(* IEC 61131-3 sources: canworks/test/cia402, 6 files *)

(* ---- drive_model.st ---- *)
(*
 * A CiA 402 drive for the ST tests (test/cia402/run.sh): the power state
 * machine (CiA 402 figure "state machine"), profile position (mode 1),
 * profile velocity (mode 3), homing (mode 6, method 35: the current
 * position is home) and the cyclic synchronous modes (8 position, 9
 * velocity, 10 torque: the set-point of each call is applied, as on one
 * SYNC), with halt (controlword bit 8) and a fault input. A mode that
 * ModesSupported (0x6502 bits) does not list is not taken: 0x6061 keeps the
 * old mode. One call is one cycle of Dt. test/drive/cia402_slave.hpp plays
 * the profile modes on a CAN bus.
 *
 * Statusword bits: 0 ready to switch on, 1 switched on, 2 operation enabled,
 * 3 fault, 4 voltage enabled, 5 quick stop (1 = not active), 6 switch on
 * disabled, 9 remote, 10 target reached, 12 set-point acknowledge / speed
 * zero / homing attained (by mode), 14 standstill (the bit the editor's
 * motion library reads as standstill).
 *)
FUNCTION_BLOCK CiA402_Drive
VAR_INPUT
	ControlWord : UINT;
	Modes : SINT;
	TargetPosition : DINT;
	ProfileVelocity : UDINT;
	TargetVelocity : DINT;
	TargetTorque : INT;
	Fault : BOOL;                (* raise a drive fault *)
	Dt : LREAL := 0.01;          (* cycle [s] *)
	ModesSupported : DWORD := DWORD#16#000003A5;  (* 0x6502: modes 1, 3, 6, 8, 9, 10 *)
	TorqueGain : LREAL := 10.0;  (* mode 10: acceleration [counts/s2] per mille of torque *)
END_VAR
VAR_OUTPUT
	StatusWord : UINT;
	ModesDisplay : SINT;
	Position : DINT;
	Velocity : DINT;
	Torque : INT;
	State : INT;                 (* 1 switch on disabled, 2 ready, 3 switched on, 4 enabled, 5 quick stop, 6 fault *)
END_VAR
VAR
	pos : LREAL;
	vel : LREAL;
	target : LREAL;
	cw : WORD;
	lastCw : WORD;
	ack : BOOL;
	homed : BOOL;
	step : LREAL;
END_VAR
	cw := UINT_TO_WORD(ControlWord);
	IF State = 0 THEN
		State := 1;
	END_IF

	(* Power state machine *)
	IF Fault AND State <> 6 THEN
		State := 6;
	ELSIF State = 6 THEN
		IF cw.7 AND NOT lastCw.7 AND NOT Fault THEN
			State := 1;
		END_IF
	ELSIF (cw AND WORD#16#0082) = WORD#16#0000 THEN
		State := 1;                                        (* disable voltage *)
	ELSIF (cw AND WORD#16#0086) = WORD#16#0002 THEN
		IF State = 4 THEN State := 5; ELSE State := 1; END_IF  (* quick stop *)
	ELSIF (cw AND WORD#16#0087) = WORD#16#0006 THEN
		State := 2;                                        (* shutdown *)
	ELSIF (cw AND WORD#16#008F) = WORD#16#0007 THEN
		IF State = 2 OR State = 4 THEN State := 3; END_IF  (* switch on / disable operation *)
	ELSIF (cw AND WORD#16#008F) = WORD#16#000F THEN
		IF State = 3 OR State = 5 THEN State := 4; END_IF  (* enable operation *)
	END_IF

	IF Modes >= SINT#1 AND Modes <= SINT#32 THEN
		IF (SHR(ModesSupported, SINT_TO_INT(Modes) - 1) AND DWORD#1) = DWORD#1 THEN
			ModesDisplay := Modes;
		END_IF
	END_IF
	Torque := 0;
	IF State <> 4 THEN
		vel := 0.0;
		ack := FALSE;
		target := pos;
	ELSIF cw.8 THEN
		vel := 0.0;                                        (* halt *)
	ELSIF ModesDisplay = 1 THEN
		IF cw.4 AND NOT lastCw.4 THEN
			IF cw.6 THEN target := target + DINT_TO_LREAL(TargetPosition);
			ELSE target := DINT_TO_LREAL(TargetPosition); END_IF
			ack := TRUE;
		ELSIF NOT cw.4 THEN
			ack := FALSE;
		END_IF
		step := UDINT_TO_LREAL(ProfileVelocity) * Dt;
		IF ABS(target - pos) <= step THEN
			vel := (target - pos) / Dt;
		ELSIF target > pos THEN
			vel := UDINT_TO_LREAL(ProfileVelocity);
		ELSE
			vel := -UDINT_TO_LREAL(ProfileVelocity);
		END_IF
	ELSIF ModesDisplay = 3 THEN
		vel := DINT_TO_LREAL(TargetVelocity);
	ELSIF ModesDisplay = 8 THEN
		vel := (DINT_TO_LREAL(TargetPosition) - pos) / Dt;   (* CSP: at the set-point after one cycle *)
		target := DINT_TO_LREAL(TargetPosition);
	ELSIF ModesDisplay = 9 THEN
		vel := DINT_TO_LREAL(TargetVelocity);
	ELSIF ModesDisplay = 10 THEN
		vel := vel + INT_TO_LREAL(TargetTorque) * TorqueGain * Dt;
		Torque := TargetTorque;
	ELSIF ModesDisplay = 6 THEN
		vel := 0.0;
		IF cw.4 AND NOT lastCw.4 THEN
			pos := 0.0;                                    (* method 35: here is home *)
			target := 0.0;
			homed := TRUE;
		ELSIF NOT cw.4 THEN
			homed := FALSE;
		END_IF
	ELSE
		vel := 0.0;
	END_IF
	pos := pos + vel * Dt;
	Position := LREAL_TO_DINT(pos);
	Velocity := LREAL_TO_DINT(vel);

	(* Statusword *)
	CASE State OF
		1: StatusWord := 16#0250;   (* switch on disabled, quick stop off, remote *)
		2: StatusWord := 16#0231;
		3: StatusWord := 16#0233;
		4: StatusWord := 16#0237;
		5: StatusWord := 16#0217;
		6: StatusWord := 16#0218;
	END_CASE
	IF vel = 0.0 THEN
		StatusWord := StatusWord OR 16#4000;                (* standstill *)
	END_IF
	IF State = 4 THEN
		IF ModesDisplay = 1 THEN
			IF ack THEN StatusWord := StatusWord OR 16#1000; END_IF
			IF pos = target THEN StatusWord := StatusWord OR 16#0400; END_IF
		ELSIF ModesDisplay = 3 THEN
			IF vel = 0.0 THEN StatusWord := StatusWord OR 16#1000; END_IF
			IF vel = DINT_TO_LREAL(TargetVelocity) THEN StatusWord := StatusWord OR 16#0400; END_IF
		ELSIF ModesDisplay = 6 THEN
			IF homed THEN StatusWord := StatusWord OR 16#1400; END_IF
		ELSIF ModesDisplay >= 8 AND ModesDisplay <= 10 THEN
			StatusWord := StatusWord OR 16#1000;            (* drive follows the command value *)
		END_IF
	END_IF
	lastCw := cw;
END_FUNCTION_BLOCK

(*
 * One bus cycle between a program and a CiA402_Drive: call it with the
 * outputs the program wrote, then copy its outputs into the program's
 * inputs (the test runner does not write VAR_IN_OUT back into a program's
 * located variables, so the test files copy them).
 *)
FUNCTION_BLOCK DriveLink
VAR_INPUT
	ControlWord : UINT;
	Modes : SINT;
	TargetPosition : DINT;
	ProfileVelocity : UDINT;
	TargetVelocity : DINT;
	TargetTorque : INT;
	Fault : BOOL;
	Lost : BOOL;                 (* the node stops answering: inputs hold, status bit FALSE *)
END_VAR
VAR_OUTPUT
	StatusWord : UINT;
	ModesDisplay : SINT;
	Position : DINT;
	Velocity : DINT;
	Torque : INT;
	Online : BOOL;
END_VAR
VAR
	Drive : CiA402_Drive;
END_VAR
	Online := NOT Lost;
	IF NOT Lost THEN
		Drive(ControlWord := ControlWord, Modes := Modes, TargetPosition := TargetPosition,
		      ProfileVelocity := ProfileVelocity, TargetVelocity := TargetVelocity, TargetTorque := TargetTorque,
		      Fault := Fault);
		StatusWord := Drive.StatusWord;
		ModesDisplay := Drive.ModesDisplay;
		Position := Drive.Position;
		Velocity := Drive.Velocity;
		Torque := Drive.Torque;
	END_IF
END_FUNCTION_BLOCK

(* ---- test_axis.st ---- *)
(*
 * The program the project generator writes for config/cia402-drive (its
 * axis `drive` and the bridge call), with the editor's PLCopen motion blocks
 * called on that axis, against the drive model. Run by test/cia402/run.sh.
 * Each cycle: the program's scan, the test's motion block calls (after the
 * bridge, as in a user program), one bus cycle. Time stands still (the test
 * runner advances it only between test statements, not inside a loop), so
 * the library's timeouts never fire; the drive model moves by its own Dt.
 *)
TEST 'MC_Power enables the drive through the CiA 402 state machine'
	VAR
		m : main;
		bus : DriveLink;
		power : MC_Power;
		status : MC_ReadStatus;
		i : INT;
		seenShutdown, seenSwitchOn : BOOL;
	END_VAR
	FOR i := 1 TO 40 DO
		m();
		power(Axis := m.drive, Enable := TRUE);
		bus(ControlWord := m.drive_Controlword, Modes := m.drive_Modes_of_operation,
		    TargetPosition := m.drive_Target_position, ProfileVelocity := m.drive_Profile_velocity,
		    TargetVelocity := m.drive_Target_velocity);
		m.drive_Statusword := bus.StatusWord;
		m.drive_Modes_of_operation_display := bus.ModesDisplay;
		m.drive_Position_actual_value := bus.Position;
		m.drive_Velocity_actual_value := bus.Velocity;
		m.drive_ok := bus.Online;
		IF (m.drive_Controlword AND 16#8F) = 16#06 THEN seenShutdown := TRUE; END_IF
		IF (m.drive_Controlword AND 16#8F) = 16#07 THEN seenSwitchOn := TRUE; END_IF
	END_FOR
	ASSERT_TRUE(seenShutdown, 'drive got Shutdown');
	ASSERT_TRUE(seenSwitchOn, 'drive got Switch on');
	ASSERT_EQ(m.drive_Controlword AND 16#8F, 16#0F, 'drive got Enable operation');
	ASSERT_EQ(bus.Drive.State, 4);
	ASSERT_TRUE(power.Status);
	ASSERT_TRUE(m.drive.bRegulatorRealState);
	status(Axis := m.drive, Enable := TRUE);
	ASSERT_TRUE(status.StandStill);
END_TEST

TEST 'MC_MoveVelocity sets mode 3 and the target velocity'
	VAR
		m : main;
		bus : DriveLink;
		power : MC_Power;
		status : MC_ReadStatus;
		i : INT;
		move : MC_MoveVelocity;
	END_VAR
	FOR i := 1 TO 80 DO
		m();
		power(Axis := m.drive, Enable := TRUE);
		move(Axis := m.drive, Execute := power.Status, Velocity := 1000.0);
		bus(ControlWord := m.drive_Controlword, Modes := m.drive_Modes_of_operation,
		    TargetPosition := m.drive_Target_position, ProfileVelocity := m.drive_Profile_velocity,
		    TargetVelocity := m.drive_Target_velocity);
		m.drive_Statusword := bus.StatusWord;
		m.drive_Modes_of_operation_display := bus.ModesDisplay;
		m.drive_Position_actual_value := bus.Position;
		m.drive_Velocity_actual_value := bus.Velocity;
		m.drive_ok := bus.Online;
	END_FOR
	ASSERT_EQ(m.drive_Modes_of_operation, 3);
	ASSERT_EQ(m.drive_Target_velocity, 1000);
	ASSERT_EQ(m.drive_Velocity_actual_value, 1000);
	ASSERT_TRUE(move.InVelocity);
	status(Axis := m.drive, Enable := TRUE);
	ASSERT_TRUE(status.ContinuousMotion);
	ASSERT_GT(m.drive.fActPosition, 100.0);
END_TEST

TEST 'MC_MoveAbsolute reaches the target in profile position'
	VAR
		m : main;
		bus : DriveLink;
		power : MC_Power;
		status : MC_ReadStatus;
		i : INT;
		move : MC_MoveAbsolute;
		busy : BOOL;
	END_VAR
	FOR i := 1 TO 200 DO
		m();
		power(Axis := m.drive, Enable := TRUE);
		move(Axis := m.drive, Execute := power.Status, Position := 500.0, Velocity := 2000.0);
		bus(ControlWord := m.drive_Controlword, Modes := m.drive_Modes_of_operation,
		    TargetPosition := m.drive_Target_position, ProfileVelocity := m.drive_Profile_velocity,
		    TargetVelocity := m.drive_Target_velocity);
		m.drive_Statusword := bus.StatusWord;
		m.drive_Modes_of_operation_display := bus.ModesDisplay;
		m.drive_Position_actual_value := bus.Position;
		m.drive_Velocity_actual_value := bus.Velocity;
		m.drive_ok := bus.Online;
		IF move.Busy THEN busy := TRUE; END_IF
		(* Done can be TRUE before the drive takes the new set-point (the
		   library checks target reached, not the set-point acknowledge), so
		   trust it only after Busy. *)
		IF busy AND move.Done THEN EXIT; END_IF
	END_FOR
	ASSERT_TRUE(busy AND move.Done);
	ASSERT_EQ(m.drive_Modes_of_operation, 1);
	ASSERT_EQ(m.drive_Target_position, 500);
	ASSERT_EQ(m.drive_Profile_velocity, 2000);
	ASSERT_EQ(bus.Drive.Position, 500);
	ASSERT_NEAR(m.drive.fActPosition, 500.0, 0.5);
END_TEST

TEST 'a drive fault is error stop and MC_Reset clears it'
	VAR
		m : main;
		bus : DriveLink;
		power : MC_Power;
		status : MC_ReadStatus;
		i : INT;
		reset : MC_Reset;
		fault : BOOL;
	END_VAR
	FOR i := 1 TO 150 DO
		fault := i >= 40 AND i < 60;
		m();
		power(Axis := m.drive, Enable := i < 60 OR i >= 100);
		reset(Axis := m.drive, Execute := i >= 70 AND i < 90);
		bus(ControlWord := m.drive_Controlword, Modes := m.drive_Modes_of_operation,
		    TargetPosition := m.drive_Target_position, ProfileVelocity := m.drive_Profile_velocity,
		    TargetVelocity := m.drive_Target_velocity, Fault := fault);
		m.drive_Statusword := bus.StatusWord;
		m.drive_Modes_of_operation_display := bus.ModesDisplay;
		m.drive_Position_actual_value := bus.Position;
		m.drive_Velocity_actual_value := bus.Velocity;
		m.drive_ok := bus.Online;
		IF i = 55 THEN
			status(Axis := m.drive, Enable := TRUE);
	ASSERT_TRUE(status.Errorstop);
			ASSERT_TRUE(m.drive.bError);
			ASSERT_TRUE(power.Error);
		END_IF
		IF i = 89 THEN
			ASSERT_TRUE(reset.Done);
			ASSERT_FALSE(m.drive.bError);
		END_IF
	END_FOR
	ASSERT_EQ(bus.Drive.State, 4);
	ASSERT_TRUE(power.Status);
END_TEST

TEST 'a lost drive (status bit FALSE) is error stop'
	VAR
		m : main;
		bus : DriveLink;
		power : MC_Power;
		status : MC_ReadStatus;
		i : INT;
	END_VAR
	FOR i := 1 TO 60 DO
		m();
		power(Axis := m.drive, Enable := TRUE);
		bus(ControlWord := m.drive_Controlword, Modes := m.drive_Modes_of_operation,
		    TargetPosition := m.drive_Target_position, ProfileVelocity := m.drive_Profile_velocity,
		    TargetVelocity := m.drive_Target_velocity, Lost := i > 40);
		m.drive_Statusword := bus.StatusWord;
		m.drive_Modes_of_operation_display := bus.ModesDisplay;
		m.drive_Position_actual_value := bus.Position;
		m.drive_Velocity_actual_value := bus.Velocity;
		m.drive_ok := bus.Online;
	END_FOR
	ASSERT_FALSE(m.drive_ok);
	ASSERT_FALSE(m.drive.bCommunication);
	status(Axis := m.drive, Enable := TRUE);
	ASSERT_TRUE(status.Errorstop);
END_TEST

(* ---- test_cyclic.st ---- *)
(*
 * The cyclic synchronous blocks (CO402_Cyclic*, library/openplc_canopen) on
 * the program the project generator writes for
 * config/cia402-drive/canopen_config_cyclic.json (task interval T#10ms, so
 * fCycleTime 0.01), against the drive model. Run by test/cia402/run.sh.
 * Each cycle: the program's scan (bridge), MC_Power and the block under
 * test, one bus cycle (one SYNC: the drive applies this cycle's set-point).
 *)
TEST 'generated lines set the cycle time'
	VAR
		m : main;
	END_VAR
	m();
	ASSERT_NEAR(m.drive.fCycleTime, 0.01, 0.0000001);
END_TEST

TEST 'CO402_CyclicVelocity selects mode 9, follows, and sends 0 when disabled'
	VAR
		m : main;
		bus : DriveLink;
		power : MC_Power;
		fault : BOOL;
		i : INT;
		csv : CO402_CyclicVelocity;
		bit3 : BOOL := TRUE;
	END_VAR
	FOR i := 1 TO 40 DO
		m();
		power(Axis := m.drive, Enable := TRUE);
		bus(ControlWord := m.drive_Controlword, Modes := m.drive_Modes_of_operation,
		    TargetPosition := m.drive_Target_position, TargetVelocity := m.drive_Target_velocity,
		    TargetTorque := m.drive_Target_torque, Fault := fault);
		m.drive_Statusword := bus.StatusWord;
		m.drive_Modes_of_operation_display := bus.ModesDisplay;
		m.drive_Position_actual_value := bus.Position;
		m.drive_Velocity_actual_value := bus.Velocity;
		m.drive_Torque_actual_value := bus.Torque;
		m.drive_ok := bus.Online;
	END_FOR
	ASSERT_TRUE(power.Status, 'powered');
	FOR i := 1 TO 30 DO
		m();
		power(Axis := m.drive, Enable := TRUE);
		csv(Axis := m.drive, Enable := TRUE, Velocity := 1000.0);
		IF (m.drive_Controlword AND 16#08) = 0 THEN bit3 := FALSE; END_IF
		bus(ControlWord := m.drive_Controlword, Modes := m.drive_Modes_of_operation,
		    TargetPosition := m.drive_Target_position, TargetVelocity := m.drive_Target_velocity,
		    TargetTorque := m.drive_Target_torque, Fault := fault);
		m.drive_Statusword := bus.StatusWord;
		m.drive_Modes_of_operation_display := bus.ModesDisplay;
		m.drive_Position_actual_value := bus.Position;
		m.drive_Velocity_actual_value := bus.Velocity;
		m.drive_Torque_actual_value := bus.Torque;
		m.drive_ok := bus.Online;
	END_FOR
	ASSERT_TRUE(bit3, 'enable operation kept while changing the mode');
	ASSERT_TRUE(csv.InSync);
	ASSERT_FALSE(csv.Error);
	ASSERT_EQ(bus.ModesDisplay, 9);
	ASSERT_EQ(m.drive_Target_velocity, 1000);
	ASSERT_EQ(bus.Velocity, 1000);
	m();
	power(Axis := m.drive, Enable := TRUE);
	csv(Axis := m.drive, Enable := FALSE, Velocity := 1000.0);
	ASSERT_EQ(m.drive.Drive.Target_Velocity, 0, 'velocity 0 in the scan Enable goes FALSE');
	ASSERT_FALSE(csv.Busy);
END_TEST

TEST 'CO402_CyclicPosition starts without a jump from the actual position'
	VAR
		m : main;
		bus : DriveLink;
		power : MC_Power;
		fault : BOOL;
		i : INT;
		csv : CO402_CyclicVelocity;
		csp : CO402_CyclicPosition;
		start : DINT;
		jump : BOOL;
		bit3 : BOOL := TRUE;
	END_VAR
	FOR i := 1 TO 40 DO
		m();
		power(Axis := m.drive, Enable := TRUE);
		bus(ControlWord := m.drive_Controlword, Modes := m.drive_Modes_of_operation,
		    TargetPosition := m.drive_Target_position, TargetVelocity := m.drive_Target_velocity,
		    TargetTorque := m.drive_Target_torque, Fault := fault);
		m.drive_Statusword := bus.StatusWord;
		m.drive_Modes_of_operation_display := bus.ModesDisplay;
		m.drive_Position_actual_value := bus.Position;
		m.drive_Velocity_actual_value := bus.Velocity;
		m.drive_Torque_actual_value := bus.Torque;
		m.drive_ok := bus.Online;
	END_FOR
	ASSERT_TRUE(power.Status, 'powered');
	(* move away from 0 in CSV first *)
	FOR i := 1 TO 50 DO
		m();
		power(Axis := m.drive, Enable := TRUE);
		csv(Axis := m.drive, Enable := TRUE, Velocity := 1000.0);
		bus(ControlWord := m.drive_Controlword, Modes := m.drive_Modes_of_operation,
		    TargetPosition := m.drive_Target_position, TargetVelocity := m.drive_Target_velocity,
		    TargetTorque := m.drive_Target_torque, Fault := fault);
		m.drive_Statusword := bus.StatusWord;
		m.drive_Modes_of_operation_display := bus.ModesDisplay;
		m.drive_Position_actual_value := bus.Position;
		m.drive_Velocity_actual_value := bus.Velocity;
		m.drive_Torque_actual_value := bus.Torque;
		m.drive_ok := bus.Online;
	END_FOR
	m();
	power(Axis := m.drive, Enable := TRUE);
	csv(Axis := m.drive, Enable := FALSE);
		bus(ControlWord := m.drive_Controlword, Modes := m.drive_Modes_of_operation,
		    TargetPosition := m.drive_Target_position, TargetVelocity := m.drive_Target_velocity,
		    TargetTorque := m.drive_Target_torque, Fault := fault);
		m.drive_Statusword := bus.StatusWord;
		m.drive_Modes_of_operation_display := bus.ModesDisplay;
		m.drive_Position_actual_value := bus.Position;
		m.drive_Velocity_actual_value := bus.Velocity;
		m.drive_Torque_actual_value := bus.Torque;
		m.drive_ok := bus.Online;
	start := bus.Position;
	ASSERT_GT(start, 400, 'the axis moved in CSV');
	FOR i := 1 TO 30 DO
		m();
		power(Axis := m.drive, Enable := TRUE);
		csp(Axis := m.drive, Enable := TRUE, Position := DINT_TO_LREAL(start), MaxVelocity := 1000.0);
		(* the outputs the bus sees are the previous scan's: count mode 8 only *)
		IF m.drive_Modes_of_operation = 8 AND ABS(m.drive_Target_position - start) > 10 THEN jump := TRUE; END_IF
		IF (m.drive_Controlword AND 16#08) = 0 THEN bit3 := FALSE; END_IF
		bus(ControlWord := m.drive_Controlword, Modes := m.drive_Modes_of_operation,
		    TargetPosition := m.drive_Target_position, TargetVelocity := m.drive_Target_velocity,
		    TargetTorque := m.drive_Target_torque, Fault := fault);
		m.drive_Statusword := bus.StatusWord;
		m.drive_Modes_of_operation_display := bus.ModesDisplay;
		m.drive_Position_actual_value := bus.Position;
		m.drive_Velocity_actual_value := bus.Velocity;
		m.drive_Torque_actual_value := bus.Torque;
		m.drive_ok := bus.Online;
	END_FOR
	ASSERT_FALSE(jump, 'no set-point away from the actual position');
	ASSERT_TRUE(bit3, 'enable operation kept while changing the mode');
	ASSERT_TRUE(csp.InSync);
	ASSERT_FALSE(csp.Error);
	ASSERT_EQ(bus.ModesDisplay, 8);
	ASSERT_EQ(m.drive_Target_position, start);
	(* follow a ramp of 5 increments per cycle, within the limit of 10 *)
	FOR i := 1 TO 20 DO
		m();
		power(Axis := m.drive, Enable := TRUE);
		csp(Axis := m.drive, Enable := TRUE, Position := DINT_TO_LREAL(start + 5 * i), MaxVelocity := 1000.0);
		bus(ControlWord := m.drive_Controlword, Modes := m.drive_Modes_of_operation,
		    TargetPosition := m.drive_Target_position, TargetVelocity := m.drive_Target_velocity,
		    TargetTorque := m.drive_Target_torque, Fault := fault);
		m.drive_Statusword := bus.StatusWord;
		m.drive_Modes_of_operation_display := bus.ModesDisplay;
		m.drive_Position_actual_value := bus.Position;
		m.drive_Velocity_actual_value := bus.Velocity;
		m.drive_Torque_actual_value := bus.Torque;
		m.drive_ok := bus.Online;
	END_FOR
	ASSERT_FALSE(csp.Error);
	ASSERT_EQ(m.drive.Drive.Target_Position, start + 100);
	ASSERT_EQ(bus.Position, start + 95, 'the drive is one scan behind (outputs go out with the next scan)');
END_TEST

TEST 'CO402_CyclicPosition refuses a step above its limit and holds the set-point'
	VAR
		m : main;
		bus : DriveLink;
		power : MC_Power;
		fault : BOOL;
		i : INT;
		csp : CO402_CyclicPosition;
	END_VAR
	FOR i := 1 TO 40 DO
		m();
		power(Axis := m.drive, Enable := TRUE);
		bus(ControlWord := m.drive_Controlword, Modes := m.drive_Modes_of_operation,
		    TargetPosition := m.drive_Target_position, TargetVelocity := m.drive_Target_velocity,
		    TargetTorque := m.drive_Target_torque, Fault := fault);
		m.drive_Statusword := bus.StatusWord;
		m.drive_Modes_of_operation_display := bus.ModesDisplay;
		m.drive_Position_actual_value := bus.Position;
		m.drive_Velocity_actual_value := bus.Velocity;
		m.drive_Torque_actual_value := bus.Torque;
		m.drive_ok := bus.Online;
	END_FOR
	ASSERT_TRUE(power.Status, 'powered');
	FOR i := 1 TO 20 DO
		m();
		power(Axis := m.drive, Enable := TRUE);
		csp(Axis := m.drive, Enable := TRUE, Position := 0.0, MaxVelocity := 1000.0);
		bus(ControlWord := m.drive_Controlword, Modes := m.drive_Modes_of_operation,
		    TargetPosition := m.drive_Target_position, TargetVelocity := m.drive_Target_velocity,
		    TargetTorque := m.drive_Target_torque, Fault := fault);
		m.drive_Statusword := bus.StatusWord;
		m.drive_Modes_of_operation_display := bus.ModesDisplay;
		m.drive_Position_actual_value := bus.Position;
		m.drive_Velocity_actual_value := bus.Velocity;
		m.drive_Torque_actual_value := bus.Torque;
		m.drive_ok := bus.Online;
	END_FOR
	ASSERT_TRUE(csp.InSync);
	m();
	power(Axis := m.drive, Enable := TRUE);
	csp(Axis := m.drive, Enable := TRUE, Position := 50.0, MaxVelocity := 1000.0);
		bus(ControlWord := m.drive_Controlword, Modes := m.drive_Modes_of_operation,
		    TargetPosition := m.drive_Target_position, TargetVelocity := m.drive_Target_velocity,
		    TargetTorque := m.drive_Target_torque, Fault := fault);
		m.drive_Statusword := bus.StatusWord;
		m.drive_Modes_of_operation_display := bus.ModesDisplay;
		m.drive_Position_actual_value := bus.Position;
		m.drive_Velocity_actual_value := bus.Velocity;
		m.drive_Torque_actual_value := bus.Torque;
		m.drive_ok := bus.Online;
	ASSERT_TRUE(csp.Error);
	ASSERT_EQ(csp.ErrorID, 3);
	ASSERT_EQ(m.drive_Target_position, 0, 'the last set-point is held');
	m();
	csp(Axis := m.drive, Enable := FALSE);
	ASSERT_FALSE(csp.Error, 'Enable FALSE clears the error');
END_TEST

TEST 'CO402_CyclicPosition reports a mode the drive does not take'
	VAR
		m : main;
		bus : DriveLink;
		power : MC_Power;
		fault : BOOL;
		i : INT;
		csp : CO402_CyclicPosition;
	END_VAR
	bus.Drive.ModesSupported := DWORD#16#00000025;  (* profile modes only *)
	FOR i := 1 TO 40 DO
		m();
		power(Axis := m.drive, Enable := TRUE);
		bus(ControlWord := m.drive_Controlword, Modes := m.drive_Modes_of_operation,
		    TargetPosition := m.drive_Target_position, TargetVelocity := m.drive_Target_velocity,
		    TargetTorque := m.drive_Target_torque, Fault := fault);
		m.drive_Statusword := bus.StatusWord;
		m.drive_Modes_of_operation_display := bus.ModesDisplay;
		m.drive_Position_actual_value := bus.Position;
		m.drive_Velocity_actual_value := bus.Velocity;
		m.drive_Torque_actual_value := bus.Torque;
		m.drive_ok := bus.Online;
	END_FOR
	ASSERT_TRUE(power.Status, 'powered');
	FOR i := 1 TO 3 DO
		m();
		power(Axis := m.drive, Enable := TRUE);
		csp(Axis := m.drive, Enable := TRUE, Position := 0.0, ModeTimeout := T#50ms);
		bus(ControlWord := m.drive_Controlword, Modes := m.drive_Modes_of_operation,
		    TargetPosition := m.drive_Target_position, TargetVelocity := m.drive_Target_velocity,
		    TargetTorque := m.drive_Target_torque, Fault := fault);
		m.drive_Statusword := bus.StatusWord;
		m.drive_Modes_of_operation_display := bus.ModesDisplay;
		m.drive_Position_actual_value := bus.Position;
		m.drive_Velocity_actual_value := bus.Velocity;
		m.drive_Torque_actual_value := bus.Torque;
		m.drive_ok := bus.Online;
	END_FOR
	ASSERT_FALSE(csp.Error, 'still waiting for the mode');
	ADVANCE_TIME(T#100ms);
	FOR i := 1 TO 3 DO
		m();
		power(Axis := m.drive, Enable := TRUE);
		csp(Axis := m.drive, Enable := TRUE, Position := 0.0, ModeTimeout := T#50ms);
		bus(ControlWord := m.drive_Controlword, Modes := m.drive_Modes_of_operation,
		    TargetPosition := m.drive_Target_position, TargetVelocity := m.drive_Target_velocity,
		    TargetTorque := m.drive_Target_torque, Fault := fault);
		m.drive_Statusword := bus.StatusWord;
		m.drive_Modes_of_operation_display := bus.ModesDisplay;
		m.drive_Position_actual_value := bus.Position;
		m.drive_Velocity_actual_value := bus.Velocity;
		m.drive_Torque_actual_value := bus.Torque;
		m.drive_ok := bus.Online;
	END_FOR
	ASSERT_TRUE(csp.Error);
	ASSERT_EQ(csp.ErrorID, 2);
END_TEST

TEST 'CO402_CyclicMoveAbsolute plans an S-curve move in CSP'
	VAR
		m : main;
		bus : DriveLink;
		power : MC_Power;
		fault : BOOL;
		i : INT;
		move : CO402_CyclicMoveAbsolute;
		last : DINT;
		step : DINT;
		maxStep : DINT;
		n : INT;
	END_VAR
	FOR i := 1 TO 40 DO
		m();
		power(Axis := m.drive, Enable := TRUE);
		bus(ControlWord := m.drive_Controlword, Modes := m.drive_Modes_of_operation,
		    TargetPosition := m.drive_Target_position, TargetVelocity := m.drive_Target_velocity,
		    TargetTorque := m.drive_Target_torque, Fault := fault);
		m.drive_Statusword := bus.StatusWord;
		m.drive_Modes_of_operation_display := bus.ModesDisplay;
		m.drive_Position_actual_value := bus.Position;
		m.drive_Velocity_actual_value := bus.Velocity;
		m.drive_Torque_actual_value := bus.Torque;
		m.drive_ok := bus.Online;
	END_FOR
	ASSERT_TRUE(power.Status, 'powered');
	FOR i := 1 TO 1000 DO
		m();
		power(Axis := m.drive, Enable := TRUE);
		move(Axis := m.drive, Execute := TRUE, Position := 10000.0, Velocity := 2000.0, Acceleration := 10000.0,
		     Jerk := 100000.0);
		step := ABS(m.drive_Target_position - last);
		IF step > maxStep THEN maxStep := step; END_IF
		last := m.drive_Target_position;
		bus(ControlWord := m.drive_Controlword, Modes := m.drive_Modes_of_operation,
		    TargetPosition := m.drive_Target_position, TargetVelocity := m.drive_Target_velocity,
		    TargetTorque := m.drive_Target_torque, Fault := fault);
		m.drive_Statusword := bus.StatusWord;
		m.drive_Modes_of_operation_display := bus.ModesDisplay;
		m.drive_Position_actual_value := bus.Position;
		m.drive_Velocity_actual_value := bus.Velocity;
		m.drive_Torque_actual_value := bus.Torque;
		m.drive_ok := bus.Online;
		IF move.Done AND n = 0 THEN n := i; END_IF
	END_FOR
	ASSERT_FALSE(move.Error);
	ASSERT_TRUE(move.Done);
	ASSERT_EQ(bus.ModesDisplay, 8);
	ASSERT_EQ(bus.Position, 10000);
	ASSERT_LE(maxStep, 21, 'no step above velocity times cycle time (20) plus rounding');
	ASSERT_GT(n, 500, 'a 10000 move at 2000/s takes over 5 s');
END_TEST

TEST 'CO402_CyclicTorque selects mode 10 and accelerates the axis'
	VAR
		m : main;
		bus : DriveLink;
		power : MC_Power;
		fault : BOOL;
		i : INT;
		cst : CO402_CyclicTorque;
	END_VAR
	FOR i := 1 TO 40 DO
		m();
		power(Axis := m.drive, Enable := TRUE);
		bus(ControlWord := m.drive_Controlword, Modes := m.drive_Modes_of_operation,
		    TargetPosition := m.drive_Target_position, TargetVelocity := m.drive_Target_velocity,
		    TargetTorque := m.drive_Target_torque, Fault := fault);
		m.drive_Statusword := bus.StatusWord;
		m.drive_Modes_of_operation_display := bus.ModesDisplay;
		m.drive_Position_actual_value := bus.Position;
		m.drive_Velocity_actual_value := bus.Velocity;
		m.drive_Torque_actual_value := bus.Torque;
		m.drive_ok := bus.Online;
	END_FOR
	ASSERT_TRUE(power.Status, 'powered');
	FOR i := 1 TO 30 DO
		m();
		power(Axis := m.drive, Enable := TRUE);
		cst(Axis := m.drive, Enable := TRUE, Torque := 100.0);
		bus(ControlWord := m.drive_Controlword, Modes := m.drive_Modes_of_operation,
		    TargetPosition := m.drive_Target_position, TargetVelocity := m.drive_Target_velocity,
		    TargetTorque := m.drive_Target_torque, Fault := fault);
		m.drive_Statusword := bus.StatusWord;
		m.drive_Modes_of_operation_display := bus.ModesDisplay;
		m.drive_Position_actual_value := bus.Position;
		m.drive_Velocity_actual_value := bus.Velocity;
		m.drive_Torque_actual_value := bus.Torque;
		m.drive_ok := bus.Online;
	END_FOR
	ASSERT_TRUE(cst.InSync);
	ASSERT_EQ(bus.ModesDisplay, 10);
	ASSERT_EQ(m.drive_Target_torque, 100);
	ASSERT_EQ(bus.Torque, 100);
	ASSERT_GT(bus.Velocity, 100, 'torque 100 at gain 10 accelerates by 1000/s2');
	m();
	cst(Axis := m.drive, Enable := FALSE);
	ASSERT_EQ(m.drive.Drive.Target_torque, 0);
END_TEST

TEST 'a drive fault stops the cyclic block with error stop'
	VAR
		m : main;
		bus : DriveLink;
		power : MC_Power;
		fault : BOOL;
		i : INT;
		csv : CO402_CyclicVelocity;
	END_VAR
	FOR i := 1 TO 40 DO
		m();
		power(Axis := m.drive, Enable := TRUE);
		bus(ControlWord := m.drive_Controlword, Modes := m.drive_Modes_of_operation,
		    TargetPosition := m.drive_Target_position, TargetVelocity := m.drive_Target_velocity,
		    TargetTorque := m.drive_Target_torque, Fault := fault);
		m.drive_Statusword := bus.StatusWord;
		m.drive_Modes_of_operation_display := bus.ModesDisplay;
		m.drive_Position_actual_value := bus.Position;
		m.drive_Velocity_actual_value := bus.Velocity;
		m.drive_Torque_actual_value := bus.Torque;
		m.drive_ok := bus.Online;
	END_FOR
	ASSERT_TRUE(power.Status, 'powered');
	FOR i := 1 TO 20 DO
		m();
		power(Axis := m.drive, Enable := TRUE);
		csv(Axis := m.drive, Enable := TRUE, Velocity := 500.0);
		bus(ControlWord := m.drive_Controlword, Modes := m.drive_Modes_of_operation,
		    TargetPosition := m.drive_Target_position, TargetVelocity := m.drive_Target_velocity,
		    TargetTorque := m.drive_Target_torque, Fault := fault);
		m.drive_Statusword := bus.StatusWord;
		m.drive_Modes_of_operation_display := bus.ModesDisplay;
		m.drive_Position_actual_value := bus.Position;
		m.drive_Velocity_actual_value := bus.Velocity;
		m.drive_Torque_actual_value := bus.Torque;
		m.drive_ok := bus.Online;
	END_FOR
	ASSERT_TRUE(csv.InSync);
	fault := TRUE;
	FOR i := 1 TO 3 DO
		m();
		power(Axis := m.drive, Enable := TRUE);
		csv(Axis := m.drive, Enable := TRUE, Velocity := 500.0);
		bus(ControlWord := m.drive_Controlword, Modes := m.drive_Modes_of_operation,
		    TargetPosition := m.drive_Target_position, TargetVelocity := m.drive_Target_velocity,
		    TargetTorque := m.drive_Target_torque, Fault := fault);
		m.drive_Statusword := bus.StatusWord;
		m.drive_Modes_of_operation_display := bus.ModesDisplay;
		m.drive_Position_actual_value := bus.Position;
		m.drive_Velocity_actual_value := bus.Velocity;
		m.drive_Torque_actual_value := bus.Torque;
		m.drive_ok := bus.Online;
	END_FOR
	ASSERT_TRUE(csv.Error);
	ASSERT_EQ(csv.ErrorID, 4);
END_TEST

TEST 'a lost drive stops the cyclic block with error stop'
	VAR
		m : main;
		bus : DriveLink;
		power : MC_Power;
		fault : BOOL;
		i : INT;
		csp : CO402_CyclicPosition;
	END_VAR
	FOR i := 1 TO 40 DO
		m();
		power(Axis := m.drive, Enable := TRUE);
		bus(ControlWord := m.drive_Controlword, Modes := m.drive_Modes_of_operation,
		    TargetPosition := m.drive_Target_position, TargetVelocity := m.drive_Target_velocity,
		    TargetTorque := m.drive_Target_torque, Fault := fault);
		m.drive_Statusword := bus.StatusWord;
		m.drive_Modes_of_operation_display := bus.ModesDisplay;
		m.drive_Position_actual_value := bus.Position;
		m.drive_Velocity_actual_value := bus.Velocity;
		m.drive_Torque_actual_value := bus.Torque;
		m.drive_ok := bus.Online;
	END_FOR
	ASSERT_TRUE(power.Status, 'powered');
	FOR i := 1 TO 20 DO
		m();
		power(Axis := m.drive, Enable := TRUE);
		csp(Axis := m.drive, Enable := TRUE, Position := 0.0);
		bus(ControlWord := m.drive_Controlword, Modes := m.drive_Modes_of_operation,
		    TargetPosition := m.drive_Target_position, TargetVelocity := m.drive_Target_velocity,
		    TargetTorque := m.drive_Target_torque, Fault := fault);
		m.drive_Statusword := bus.StatusWord;
		m.drive_Modes_of_operation_display := bus.ModesDisplay;
		m.drive_Position_actual_value := bus.Position;
		m.drive_Velocity_actual_value := bus.Velocity;
		m.drive_Torque_actual_value := bus.Torque;
		m.drive_ok := bus.Online;
	END_FOR
	ASSERT_TRUE(csp.InSync);
	m.drive_ok := FALSE;
	m();
	power(Axis := m.drive, Enable := TRUE);
	csp(Axis := m.drive, Enable := TRUE, Position := 0.0);
	ASSERT_TRUE(csp.Error);
	ASSERT_EQ(csp.ErrorID, 4);
END_TEST

(* ---- test_cyclic_demo.st ---- *)
(*
 * config/cia402-drive/drive_cyclic_demo.st against the drive model, with
 * the cyclic blocks of the packaged openplc_canopen library. Run by
 * test/cia402/run.sh. The demo counts its times in task cycles, so one loop
 * pass is one 10 ms cycle and one SYNC.
 *)
TEST 'the cyclic demo powers on, homes, moves in CSP, runs in CSV and steps in CST'
	VAR
		m : main;
		bus : DriveLink;
		f : BOOL;
		i : INT;
		last : DINT;
		jump : DINT;
		maxStep : DINT;
		peak : DINT;
		seen30 : BOOL;
		seen40 : BOOL;
	END_VAR
	FOR i := 1 TO 3000 DO
		last := m.drive_Target_position;
		m();
		bus(ControlWord := m.drive_Controlword, Modes := m.drive_Modes_of_operation,
		    TargetPosition := m.drive_Target_position, TargetVelocity := m.drive_Target_velocity,
		    TargetTorque := m.drive_Target_torque, Fault := f);
		m.drive_Statusword := bus.StatusWord;
		m.drive_Modes_of_operation_display := bus.ModesDisplay;
		m.drive_Position_actual_value := bus.Position;
		m.drive_Velocity_actual_value := bus.Velocity;
		m.drive_Torque_actual_value := bus.Torque;
		m.drive_ok := bus.Online;
		IF m.step = 20 AND m.drive_Modes_of_operation = 8 THEN
			jump := ABS(m.drive_Target_position - last);
			IF jump > maxStep THEN maxStep := jump; END_IF
		END_IF
		IF m.step = 30 THEN
			seen30 := TRUE;
			ASSERT_EQ(bus.Drive.Position >= 999, TRUE);
		END_IF
		IF m.step = 40 THEN
			seen40 := TRUE;
			IF ABS(bus.Velocity) > peak THEN peak := ABS(bus.Velocity); END_IF
		END_IF
		IF m.step = 50 THEN EXIT; END_IF
	END_FOR
	ASSERT_EQ(m.step, 50);
	ASSERT_EQ(m.errors, 0);
	ASSERT_TRUE(seen30 AND seen40);
	(* 500 u/s at 10 ms: at most 5 units per SYNC *)
	ASSERT_TRUE(maxStep > 0 AND maxStep <= 6, 'CSP steps within the velocity');
	(* 0.3 s at 20 per mille x gain 10: 60 u/s *)
	ASSERT_TRUE(peak >= 50 AND peak <= 70, 'CST torque step');
	FOR i := 1 TO 20 DO
		m();
		bus(ControlWord := m.drive_Controlword, Modes := m.drive_Modes_of_operation,
		    TargetPosition := m.drive_Target_position, TargetVelocity := m.drive_Target_velocity,
		    TargetTorque := m.drive_Target_torque, Fault := f);
		m.drive_Statusword := bus.StatusWord;
		m.drive_Modes_of_operation_display := bus.ModesDisplay;
		m.drive_Position_actual_value := bus.Position;
		m.drive_Velocity_actual_value := bus.Velocity;
		m.drive_Torque_actual_value := bus.Torque;
		m.drive_ok := bus.Online;
	END_FOR
	ASSERT_EQ(bus.ModesDisplay, 9);
	ASSERT_EQ(m.drive_Target_velocity, 0);
	ASSERT_TRUE(m.csv.InSync);
END_TEST

TEST 'a fault during the cyclic demo is reset and the sequence starts again'
	VAR
		m : main;
		bus : DriveLink;
		f : BOOL;
		i : INT;
	END_VAR
	FOR i := 1 TO 3000 DO
		f := FALSE;
		IF m.step = 30 AND m.errors = 0 THEN f := TRUE; END_IF
		m();
		bus(ControlWord := m.drive_Controlword, Modes := m.drive_Modes_of_operation,
		    TargetPosition := m.drive_Target_position, TargetVelocity := m.drive_Target_velocity,
		    TargetTorque := m.drive_Target_torque, Fault := f);
		m.drive_Statusword := bus.StatusWord;
		m.drive_Modes_of_operation_display := bus.ModesDisplay;
		m.drive_Position_actual_value := bus.Position;
		m.drive_Velocity_actual_value := bus.Velocity;
		m.drive_Torque_actual_value := bus.Torque;
		m.drive_ok := bus.Online;
		IF m.step = 50 THEN EXIT; END_IF
	END_FOR
	ASSERT_EQ(m.errors, 1);
	ASSERT_EQ(m.step, 50);
	ASSERT_FALSE(m.csv.Error);
END_TEST

(* ---- test_demo.st ---- *)
(*
 * config/cia402-drive/drive_demo.st against the drive model. Run by
 * test/cia402/run.sh. Time stands still inside a loop (the test runner
 * advances it only between statements), so the 2 s run step is crossed with
 * ADVANCE_TIME between two loops.
 *)
TEST 'the demo powers on, homes, moves, runs and halts'
	VAR
		m : main;
		bus : DriveLink;
		i : INT;
	END_VAR
	FOR i := 1 TO 400 DO
		m();
		bus(ControlWord := m.drive_Controlword, Modes := m.drive_Modes_of_operation,
		    TargetPosition := m.drive_Target_position, ProfileVelocity := m.drive_Profile_velocity,
		    TargetVelocity := m.drive_Target_velocity);
		m.drive_Statusword := bus.StatusWord;
		m.drive_Modes_of_operation_display := bus.ModesDisplay;
		m.drive_Position_actual_value := bus.Position;
		m.drive_Velocity_actual_value := bus.Velocity;
		m.drive_ok := bus.Online;
		IF m.step = 30 THEN EXIT; END_IF
	END_FOR
	ASSERT_EQ(m.step, 30);
	ASSERT_TRUE(m.home.Done OR m.moveAbs.Done);
	ASSERT_EQ(bus.Drive.Position, 1000);
	FOR i := 1 TO 50 DO
		m();
		bus(ControlWord := m.drive_Controlword, Modes := m.drive_Modes_of_operation,
		    TargetPosition := m.drive_Target_position, ProfileVelocity := m.drive_Profile_velocity,
		    TargetVelocity := m.drive_Target_velocity);
		m.drive_Statusword := bus.StatusWord;
		m.drive_Modes_of_operation_display := bus.ModesDisplay;
		m.drive_Position_actual_value := bus.Position;
		m.drive_Velocity_actual_value := bus.Velocity;
		m.drive_ok := bus.Online;
	END_FOR
	ASSERT_EQ(m.drive_Modes_of_operation, 3);
	ASSERT_EQ(bus.Velocity, 200);
	ADVANCE_TIME(2100000000);
	FOR i := 1 TO 100 DO
		m();
		bus(ControlWord := m.drive_Controlword, Modes := m.drive_Modes_of_operation,
		    TargetPosition := m.drive_Target_position, ProfileVelocity := m.drive_Profile_velocity,
		    TargetVelocity := m.drive_Target_velocity);
		m.drive_Statusword := bus.StatusWord;
		m.drive_Modes_of_operation_display := bus.ModesDisplay;
		m.drive_Position_actual_value := bus.Position;
		m.drive_Velocity_actual_value := bus.Velocity;
		m.drive_ok := bus.Online;
		IF m.step = 50 THEN EXIT; END_IF
	END_FOR
	ASSERT_EQ(m.step, 50);
	ASSERT_EQ(bus.Velocity, 0);
	ASSERT_TRUE(m.status.StandStill);
END_TEST

TEST 'a fault during the demo is reset and the sequence starts again'
	VAR
		m : main;
		bus : DriveLink;
		i : INT;
	END_VAR
	VAR
		f : BOOL;
	END_VAR
	FOR i := 1 TO 600 DO
		f := i >= 60 AND i < 70;
		m();
		bus(ControlWord := m.drive_Controlword, Modes := m.drive_Modes_of_operation,
		    TargetPosition := m.drive_Target_position, ProfileVelocity := m.drive_Profile_velocity,
		    TargetVelocity := m.drive_Target_velocity, Fault := f);
		m.drive_Statusword := bus.StatusWord;
		m.drive_Modes_of_operation_display := bus.ModesDisplay;
		m.drive_Position_actual_value := bus.Position;
		m.drive_Velocity_actual_value := bus.Velocity;
		m.drive_ok := bus.Online;
		IF i = 65 THEN
			ASSERT_EQ(m.step, 90);
		END_IF
		IF i > 70 AND m.step = 30 THEN EXIT; END_IF
	END_FOR
	ASSERT_EQ(m.step, 30);
	ASSERT_EQ(bus.Drive.Position, 1000);
END_TEST

(* ---- test_scaling.st ---- *)
(*
 * The program generated from config/cia402-drive with "scale_numerator": 10
 * (10 increments per technical unit), against the drive model. Run by
 * test/cia402/run.sh.
 *)
TEST 'scaling from the config converts technical units to increments'
	VAR
		m : main;
		bus : DriveLink;
		power : MC_Power;
		status : MC_ReadStatus;
		i : INT;
		move : MC_MoveVelocity;
	END_VAR
	FOR i := 1 TO 80 DO
		m();
		power(Axis := m.drive, Enable := TRUE);
		move(Axis := m.drive, Execute := power.Status, Velocity := 25.0);
		bus(ControlWord := m.drive_Controlword, Modes := m.drive_Modes_of_operation,
		    TargetPosition := m.drive_Target_position, ProfileVelocity := m.drive_Profile_velocity,
		    TargetVelocity := m.drive_Target_velocity);
		m.drive_Statusword := bus.StatusWord;
		m.drive_Modes_of_operation_display := bus.ModesDisplay;
		m.drive_Position_actual_value := bus.Position;
		m.drive_Velocity_actual_value := bus.Velocity;
		m.drive_ok := bus.Online;
	END_FOR
	ASSERT_EQ(m.drive_Target_velocity, 250);
	ASSERT_NEAR(m.drive.fActVelocity, 25.0, 0.01);
END_TEST
